// TIA Portal V18 export
DATA_BLOCK "deleteddb"   // DB60
{ S7_Optimized_Access := 'TRUE' }
VERSION : 0.1
// stored: AutoNumber true, DBAccessibleFromOPCUA true, IsOnlyStoredInLoadMemory false, IsRetainMemResEnabled false, IsWriteProtectedInAS false, MemoryReserve 100
   VAR
      target : Real;
      pos : Real;
      delta : Real;
      prec_au : Real;
      dist_stop : Real;
      arrived : Bool;
      stop_now : Bool;
      distance : Real;
   END_VAR
BEGIN
END_DATA_BLOCK
